SUBAPPLICATION Uebung_012k_sub (* String Input und Speichern INI mit Subapp *)
  (* Standard: 61499-2; Description: Copyright (c) 2023 Meisterschulen am Ostbahnhof This program and the accompanying materials are made available under the terms of the Eclipse Public License 2.0 which is available at https://www.eclipse.org/legal/epl-2.0/ SPDX-License-Identifier: EPL-2.0 *)
  (* Version 1.0, 2023-10-31, Franz Höpfinger, Meisterschulen am Ostbahnhof, initial API and implementation and/or initial documentation *)
  PACKAGE Uebungen;
  IMPORT isobus::UT::Q::const::IDs::ID_NULL;
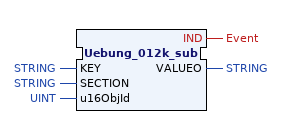
  EVENT_OUTPUT
    IND;
  END_EVENT
  VAR_INPUT
    KEY : STRING;
    SECTION : STRING;
    u16ObjId : UINT := ID_NULL;
  END_VAR
  VAR_OUTPUT
    VALUEO : STRING;
  END_VAR
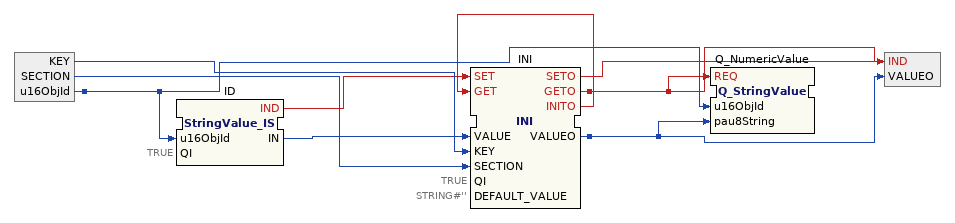
  FBS
    ID : isobus::UT::io::StringValue::StringValue_IS(QI := TRUE);
    INI : eclipse4diac::storage::INI(QI := TRUE, DEFAULT_VALUE := STRING#'');
    Q_NumericValue : isobus::UT::Q::Q_StringValue;
  END_FBS
  EVENT_CONNECTIONS
    ID.IND TO INI.SET;
    INI.SETO TO IND;
    INI.GETO TO Q_NumericValue.REQ;
    INI.GETO TO IND;
    INI.INITO TO INI.GET;
  END_CONNECTIONS
  DATA_CONNECTIONS
    ID.IN TO INI.VALUE;
    u16ObjId TO Q_NumericValue.u16ObjId;
    KEY TO INI.KEY;
    INI.VALUEO TO Q_NumericValue.pau8String;
    INI.VALUEO TO VALUEO;
    u16ObjId TO ID.u16ObjId;
    SECTION TO INI.SECTION;
  END_CONNECTIONS
END_SUBAPPLICATION
